// Mitsubishi GX Works2 project: z16   PLC: Q02/Q02H

PROGRAM MAIN
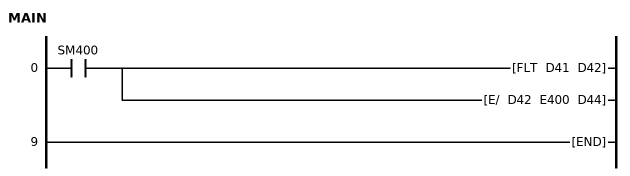
0     LD      SM400
      FLT     D41 D42
      E/      D42 E400 D44
9     END
END_PROGRAM
